FUNCTION_BLOCK EL3692
VAR
	_io : EL3692_Data;
	{attribute addProperty Name "WcState"}
	_wcState : WcStateInputToggle;
	{attribute addProperty Name "Info data"}
	_infoData : InfoDataAds;
END_VAR

PROPERTY IO : REFERENCE TO EL3692_Data
GET
IO REF= _io;
END_GET
END_PROPERTY

PROPERTY WcState : REFERENCE TO WcStateInputToggle
GET
WcState REF= _wcState;
END_GET
END_PROPERTY

END_FUNCTION_BLOCK

(* stored: Version 1.1.0.1, ProductVersion 3.1.4024.9
   POU EL3692: Id {b79d3e60-94d9-0773-1124-921aac75faa8}, SpecialFunc None
   Property IO: Id {1da20d02-b90f-0339-0ee7-08e21e71fdac}
   Get Get: Id {722f0b99-4fcc-03c8-0fc6-174f9288db5f}
   Property WcState: Id {4f22e249-12b7-01d3-3102-e7795eb2644d}
   Get Get: Id {7df7f459-794f-01bf-34bb-0c29fd5d2cf7} *)
